// Mitsubishi GX Works2 project: BookEX6_39 Special Function   PLC: Q13UDV

// global labels: Global
VAR_GLOBAL
  bVar0 AT M5000 : BOOL;
  abArray0 AT M5010 : ARRAY [0..49] OF BOOL;
  sStr0 AT D5000 : STRING[199];
  sStr1 AT D5100 : STRING[199];
  sStr2 AT D5200 : STRING[199];
  sStr3 AT D5300 : STRING[199];
  sStr4 AT D5400 : STRING[199];
  sStr5 AT D5500 : STRING[199];
  sStr6 AT D5600 : STRING[199];
  sStr7 AT D5700 : STRING[199];
  sStr8 AT D5800 : STRING[199];
  sStr9 AT D5900 : STRING[199];
  iVar0 AT D4500 : INT;
  iVar1 AT D4501 : INT;
  iVar2 AT D4502 : INT;
  iVar3 AT D4503 : INT;
  iVar4 AT D4504 : INT;
  iVar5 AT D4505 : INT;
  iVar6 AT D4506 : INT;
  iVar7 AT D4507 : INT;
  iVar8 AT D4508 : INT;
  iVar9 AT D4509 : INT;
  dVar0 AT D4510 : DINT;
  dVar1 AT D4512 : DINT;
  dVar2 AT D4514 : DINT;
  dVar3 AT D4516 : DINT;
  dVar4 AT D4518 : DINT;
  dVar5 AT D4520 : DINT;
  dVar6 AT D4522 : DINT;
  dVar7 AT D4524 : DINT;
  dVar8 AT D4526 : DINT;
  dVar9 AT D4528 : DINT;
  wVar0 AT D4530 : WORD;
  wVar1 AT D4531 : WORD;
  wVar2 AT D4532 : WORD;
  wVar3 AT D4533 : WORD;
  wVar4 AT D4534 : WORD;
  wVar5 AT D4535 : WORD;
  wVar6 AT D4536 : WORD;
  wVar7 AT D4537 : WORD;
  wVar8 AT D4538 : WORD;
  wVar9 AT D4539 : WORD;
  dwVar0 AT D4540 : DWORD;
  dwVar1 AT D4542 : DWORD;
  dwVar2 AT D4544 : DWORD;
  dwVar3 AT D4546 : DWORD;
  dwVar4 AT D4548 : DWORD;
  dwVar5 AT D4550 : DWORD;
  dwVar6 AT D4552 : DWORD;
  dwVar7 AT D4554 : DWORD;
  dwVar8 AT D4556 : DWORD;
  dwVar9 AT D4558 : DWORD;
  fsVar0 AT D4560 : REAL;
  fsVar1 AT D4562 : REAL;
  fsVar2 AT D4564 : REAL;
  fsVar3 AT D4566 : REAL;
  fsVar4 AT D4568 : REAL;
  fsVar5 AT D4570 : REAL;
  fsVar6 AT D4572 : REAL;
  fsVar7 AT D4574 : REAL;
  fsVar8 AT D4576 : REAL;
  fsVar9 AT D4578 : REAL;
  fdVar0 AT D4580 : LREAL;
  tTime0 AT D4620 : TIME;
  tTime1 AT D4622 : TIME;
  tTime2 AT D4624 : TIME;
  tTime3 AT D4626 : TIME;
  tTime4 AT D4628 : TIME;
  tTime5 AT D4630 : TIME;
  tTime6 AT D4632 : TIME;
  tTime7 AT D4634 : TIME;
  tTime8 AT D4636 : TIME;
  tTime9 AT D4638 : TIME;
  tTime10 AT D4640 : TIME;
  bVar1 AT M5001 : BOOL;
  bVar2 AT M5002 : BOOL;
  bVar3 AT M5003 : BOOL;
  bVar4 AT M5004 : BOOL;
  bVar5 AT M5005 : BOOL;
  bVar6 AT M5006 : BOOL;
  bVar7 AT M5007 : BOOL;
  bVar8 AT M5008 : BOOL;
  bVar9 AT M5009 : BOOL;
  abArray1 AT M5060 : ARRAY [0..49] OF BOOL;
  abArray2 AT M5110 : ARRAY [0..49] OF BOOL;
  abArray3 AT M5160 : ARRAY [0..49] OF BOOL;
  abArray4 AT M5210 : ARRAY [0..49] OF BOOL;
  abArray5 AT M5260 : ARRAY [0..49] OF BOOL;
  abArray6 AT M5310 : ARRAY [0..49] OF BOOL;
  abArray7 AT M5360 : ARRAY [0..49] OF BOOL;
  abArray8 AT M5410 : ARRAY [0..49] OF BOOL;
  abArray9 AT M5460 : ARRAY [0..49] OF BOOL;
  fdVar1 AT D4584 : LREAL;
  fdVar2 AT D4588 : LREAL;
  fdVar3 AT D4592 : LREAL;
  fdVar4 AT D4596 : LREAL;
  fdVar5 AT D4600 : LREAL;
  fdVar6 AT D4604 : LREAL;
  fdVar7 AT D4608 : LREAL;
  fdVar8 AT D4612 : LREAL;
  fdVar9 AT D4616 : LREAL;
  afsPen0 AT D2000 : ARRAY [0..499] OF REAL;
  afsPen1 AT D3000 : ARRAY [0..499] OF REAL;
  adwD10 AT D10 : ARRAY [0..9] OF DWORD;
  awD10 AT D10 : ARRAY [0..19] OF WORD;
  aiD10 AT D10 : ARRAY [0..19] OF INT;
  abM10 AT M10 : ARRAY [0..19] OF BOOL;
END_VAR
// user libraries (not included): HMI

FUNCTION DEG2RAD
VAR_INPUT
  fs_Deg : REAL;
END_VAR
VAR
  fsTemp : REAL;
  fs2Phi : REAL;
  dFloor : DINT;
END_VAR
VAR CONSTANT
  Phi : REAL := 3.141592653;
END_VAR
;
fsTemp := 0.0174532925199433 * fs_Deg;
fs2Phi := Phi * 2.0;
dFloor := REAL_TO_DINT(fsTemp / fs2Phi );
Deg2Rad := fsTemp;
END_FUNCTION

FUNCTION_BLOCK GenLotto
VAR_OUTPUT
  i_Lotto1 : INT;
  i_Lotto2 : INT;
  i_Lotto3 : INT;
  i_Lotto4 : INT;
  i_Lotto5 : INT;
  i_Lotto6 : INT;
END_VAR
VAR
  fbGenRandom : GenRandom;
  ix : INT;
  iy : INT;
  aiNo : ARRAY [0..5] OF INT;
  aiSNo : ARRAY [0..1] OF INT;
  idx : INT;
  bSRes : BOOL;
  aiSNo1 : ARRAY [0..1] OF INT;
  dNo : DINT;
  iz : INT;
END_VAR
;
FOR ix := 0 TO 5 DO 
	aiNo[ix] := 0;
END_FOR;
idx := 0;

REPEAT
	fbGenRandom(EN := TRUE, d_Low := 1, d_High := 45);
	dNo := fbGenRandom.d_Out;
	iy := DINT_TO_INT(dNo);
	SER(TRUE, iy, aiNo[0], 6, aiSNo);
	IF aiSNo[1] = 0 THEN
		aiNo[idx] := iy;
		idx := idx + 1;
	END_IF;
	UNTIL idx > 5
END_REPEAT;	
(* Sort *)
FOR ix := 0 TO 4 DO 
	FOR iy := 0 TO 4 DO 
		IF aiNo[iy] > aiNo[iy+1] THEN
			iz := aiNo[iy];
			aiNo[iy] := aiNo[iy+1];
			aiNo[iy+1] := iz;
		END_IF;
	END_FOR;
END_FOR;

i_Lotto1 := aiNo[0];
i_Lotto2 := aiNo[1];
i_Lotto3 := aiNo[2];
i_Lotto4 := aiNo[3];
i_Lotto5 := aiNo[4];
i_Lotto6 := aiNo[5];
END_FUNCTION_BLOCK

FUNCTION_BLOCK GenRandom
VAR_INPUT
  d_Low : DINT;
  d_High : DINT;
END_VAR
VAR
  dwTemp1 : DWORD;
END_VAR
VAR_OUTPUT
  d_Out : DINT;
END_VAR
VAR
  dLast : DINT;
  iTime : ARRAY [0..7] OF INT;
  dwTemp2 : DWORD;
  dwTemp3 : DWORD;
END_VAR
;
S_DATERD(TRUE, iTime);
dwTemp1 := DINT_TO_DWORD(INT_TO_DINT(iTime[5]) * 10000 + INT_TO_DINT(iTime[6]) * 1000 + INT_TO_DINT(iTime[7]));
dwTemp2 := SHL(dwTemp1, 15) XOR dwTemp1;
dwTemp2 := SHL(dwTemp2, 13) XOR dwTemp2;
dwTemp2 := SHR(dwTemp2, 17) XOR dwTemp2;
dLast := DWORD_TO_DINT(SHL(dwTemp2, 5) XOR dwTemp2);
d_Out := ABS(dLast MOD (d_High - d_Low + 1)) + d_Low;
END_FUNCTION_BLOCK

FUNCTION_BLOCK GenWave
VAR_INPUT
  t_Period : TIME;
  dDelay : DINT;  (* % *)
  fs_Amp : REAL;
  fs_Offset : REAL;
END_VAR
VAR_OUTPUT
  b_Q : BOOL;
  i_OutV : INT;
END_VAR
VAR
  fsTemp : REAL;
  fsTemp1 : REAL;
  tLast : TIME;
  tPast : TIME;
  tCurr : TIME;
  tMulTime : TIME;
  tShift : TIME;
  dSftTime : DINT;
  bInit : BOOL;
  qTemp : BOOL;
END_VAR
VAR CONSTANT
  PI2 : REAL := 6.283185;
END_VAR
VAR
  fbTON : TON;
END_VAR
VAR_INPUT
  i_Type : INT;
END_VAR
VAR
  dMulTime : DINT;
  dHalfPeriod : DINT;
END_VAR
;
fbTON(IN := NOT qTemp, PT := T#30m, Q:= qTemp, ET := tPast);
tCurr := tPast - tLast;

IF NOT bInit THEN
	bInit := TRUE;
	tLast := tCurr;
	tCurr := T#0s;
END_IF;

IF tCurr >= t_Period THEN
	tLast := tLast + t_Period;
	tCurr := tCurr - t_Period;
END_IF;

CASE i_Type OF 
	0 : (* SIN *)
		IF t_Period > T#0s THEN
			dSftTime := TIME_TO_DINT(t_Period) * dDelay / 100;
			tShift := DINT_TO_TIME(dSftTime);
			tMulTime := tCurr - tShift;
			fsTemp1 := PI2 * DINT_TO_REAL(TIME_TO_DINT(tMulTime)) / DINT_TO_REAL(TIME_TO_DINT(t_Period));
			SIN(TRUE, fsTemp1, fsTemp);
		ELSE
			fsTemp := 0.0;
		END_IF;
	1 : (* SQUARE *)
		IF t_Period > T#0s THEN
			dMulTime := TIME_TO_DINT(tCurr);
			dHalfPeriod := TIME_TO_DINT(t_Period) / 2;
			IF dMulTime < dHalfPeriod THEN
				fsTemp := 1.0;
			ELSE
				fsTemp := -1.0;
			END_IF;
		ELSE
			fsTemp := 0.0;
		END_IF; 
	2 : (* SAW *)
		IF t_Period > T#0s THEN
			fsTemp := DINT_TO_REAL(TIME_TO_DINT(tCurr) * 2) / DINT_TO_REAL(TIME_TO_DINT(t_Period)) - 1.0;
		ELSE
			fsTemp := 0.0;
		END_IF;
END_CASE;
i_OutV := REAL_TO_INT(fs_Amp * fsTemp * 0.5  + fs_Offset);
b_Q := i_OutV < 0;
END_FUNCTION_BLOCK

FUNCTION RAD2DEG
VAR_INPUT
  fs_Rad : REAL;
END_VAR
VAR
  fsTemp : REAL;
  fs2Phi : REAL;
  dFloor : DINT;
END_VAR
VAR CONSTANT
  Phi : REAL := 3.141592653;
END_VAR
;
fsTemp := 57.29577951308232 * fs_Rad;
dFloor := REAL_TO_DINT(fsTemp / 360.0);
Rad2Deg := fsTemp;
END_FUNCTION

PROGRAM ExASIN
VAR
  awBCD1 : ARRAY [0..2] OF WORD;
  Mov4WORD_1 : Mov4WORD;
  Mov4WORD_2 : Mov4WORD;
  Mov4WORD_3 : Mov4WORD;
  awBCD2 : ARRAY [0..2] OF WORD;
  awBCD3 : ARRAY [0..2] OF WORD;
  Mov4WORD_4 : Mov4WORD;
  awBCD4 : ARRAY [0..2] OF WORD;
  awBCD5 : ARRAY [0..2] OF WORD;
END_VAR
(* structured ladder/FBD written out as ST: instructions are called as NAME(EN, inputs, outputs); _pN, _eN, _tN stand for wires *)
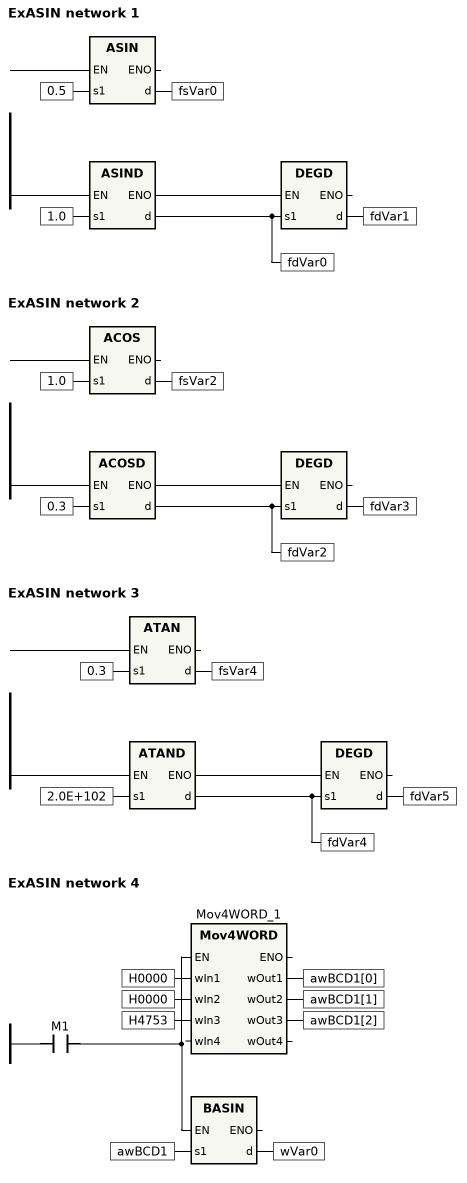
(* network 1 *)
ASIN(TRUE, 0.5, fsVar0);
_e1 := ASIND(TRUE, 1.0, fdVar0);
DEGD(_e1, fdVar0, fdVar1);
(* network 2 *)
ACOS(TRUE, 1.0, fsVar2);
_e1 := ACOSD(TRUE, 0.3, fdVar2);
DEGD(_e1, fdVar2, fdVar3);
(* network 3 *)
ATAN(TRUE, 0.3, fsVar4);
_e1 := ATAND(TRUE, 2.0E+102, fdVar4);
DEGD(_e1, fdVar4, fdVar5);
(* network 4 *)
Mov4WORD_1(EN := M1, wIn1 := H0000, wIn2 := H0000, wIn3 := H4753, wOut1 => awBCD1[0], wOut2 => awBCD1[1], wOut3 => awBCD1[2]);
BASIN(M1, awBCD1, wVar0);
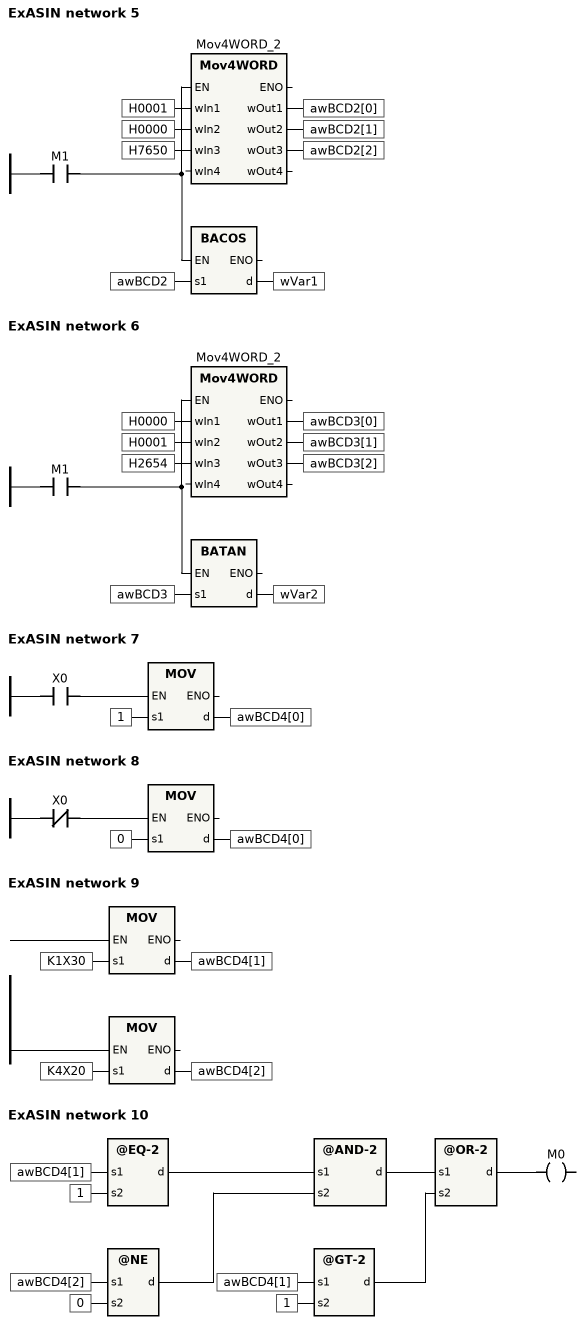
(* network 5 *)
Mov4WORD_2(EN := M1, wIn1 := H0001, wIn2 := H0000, wIn3 := H7650, wOut1 => awBCD2[0], wOut2 => awBCD2[1], wOut3 => awBCD2[2]);
BACOS(M1, awBCD2, wVar1);
(* network 6 *)
Mov4WORD_2(EN := M1, wIn1 := H0000, wIn2 := H0001, wIn3 := H2654, wOut1 => awBCD3[0], wOut2 => awBCD3[1], wOut3 => awBCD3[2]);
BATAN(M1, awBCD3, wVar2);
(* network 7 *)
MOV(X0, 1, awBCD4[0]);
(* network 8 *)
MOV(NOT X0, 0, awBCD4[0]);
(* network 9 *)
MOV(TRUE, K1X30, awBCD4[1]);
MOV(TRUE, K4X20, awBCD4[2]);
(* network 10 *)
M0 := @OR-2(@AND-2(@EQ-2(awBCD4[1], 1), @NE(awBCD4[2], 0)), @GT-2(awBCD4[1], 1));
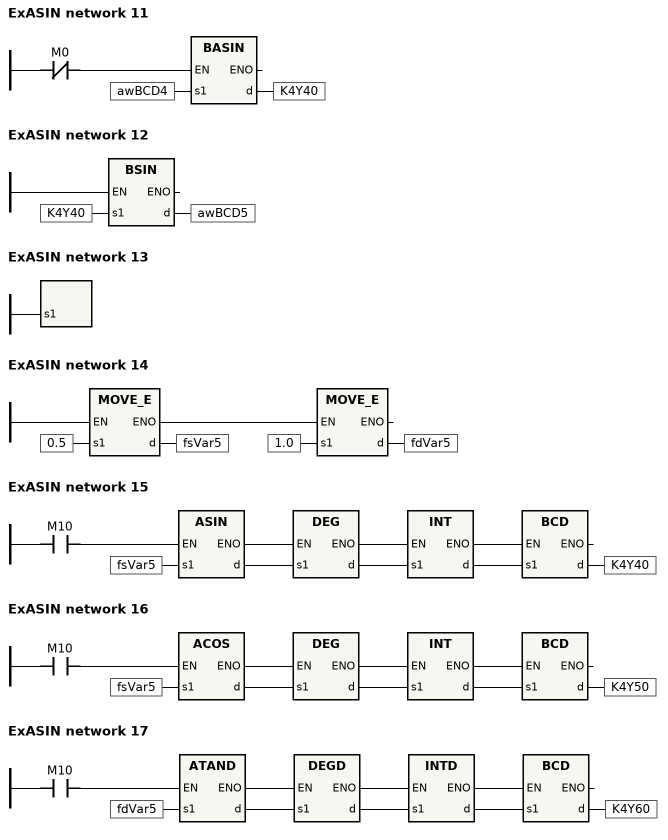
(* network 11 *)
BASIN(NOT M0, awBCD4, K4Y40);
(* network 12 *)
BSIN(TRUE, K4Y40, awBCD5);
(* network 13 *)
(* element kind 10  <- TRUE *)
(* network 14 *)
_e1 := MOVE_E(TRUE, 0.5, fsVar5);
MOVE_E(_e1, 1.0, fdVar5);
(* network 15 *)
_e2 := ASIN(M10, fsVar5, _t1);
_e4 := DEG(_e2, _t1, _t3);
_e6 := INT(_e4, _t3, _t5);
BCD(_e6, _t5, K4Y40);
(* network 16 *)
_e2 := ACOS(M10, fsVar5, _t1);
_e4 := DEG(_e2, _t1, _t3);
_e6 := INT(_e4, _t3, _t5);
BCD(_e6, _t5, K4Y50);
(* network 17 *)
_e2 := ATAND(M10, fdVar5, _t1);
_e4 := DEGD(_e2, _t1, _t3);
_e6 := INTD(_e4, _t3, _t5);
BCD(_e6, _t5, K4Y60);
END_PROGRAM

PROGRAM ExDEG_RAD
VAR
  fsLVar0 : REAL;
  fsLVar1 : REAL;
  fsLVar2 : REAL;
  fsLVar3 : REAL;
  fsLVar4 : REAL;
  fsLVar5 : REAL;
  fsLVar6 : REAL;
  fsLVar7 : REAL;
  fsLVar8 : REAL;
  fsLVar9 : REAL;
END_VAR
(* structured ladder/FBD written out as ST: instructions are called as NAME(EN, inputs, outputs); _pN, _eN, _tN stand for wires *)
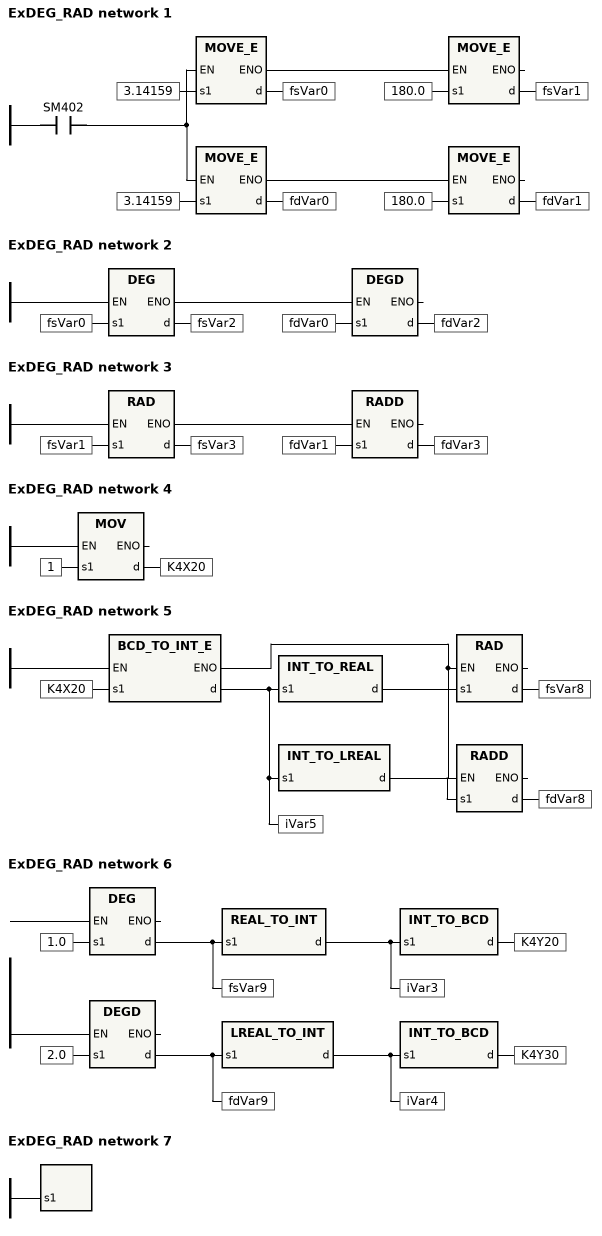
(* network 1 *)
_e1 := MOVE_E(SM402, 3.14159, fsVar0);
MOVE_E(_e1, 180.0, fsVar1);
_e2 := MOVE_E(SM402, 3.14159, fdVar0);
MOVE_E(_e2, 180.0, fdVar1);
(* network 2 *)
_e1 := DEG(TRUE, fsVar0, fsVar2);
DEGD(_e1, fdVar0, fdVar2);
(* network 3 *)
_e1 := RAD(TRUE, fsVar1, fsVar3);
RADD(_e1, fdVar1, fdVar3);
(* network 4 *)
MOV(TRUE, 1, K4X20);
(* network 5 *)
_e1 := BCD_TO_INT_E(TRUE, K4X20, iVar5);
RAD(_e1, INT_TO_REAL(iVar5), fsVar8);
RADD(_e1, INT_TO_LREAL(iVar5), fdVar8);
(* network 6 *)
DEG(TRUE, 1.0, fsVar9);
_p1 := REAL_TO_INT(fsVar9);
iVar3 := _p1;
K4Y20 := INT_TO_BCD(_p1);
DEGD(TRUE, 2.0, fdVar9);
_p2 := LREAL_TO_INT(fdVar9);
iVar4 := _p2;
K4Y30 := INT_TO_BCD(_p2);
(* network 7 *)
(* element kind 10  <- TRUE *)
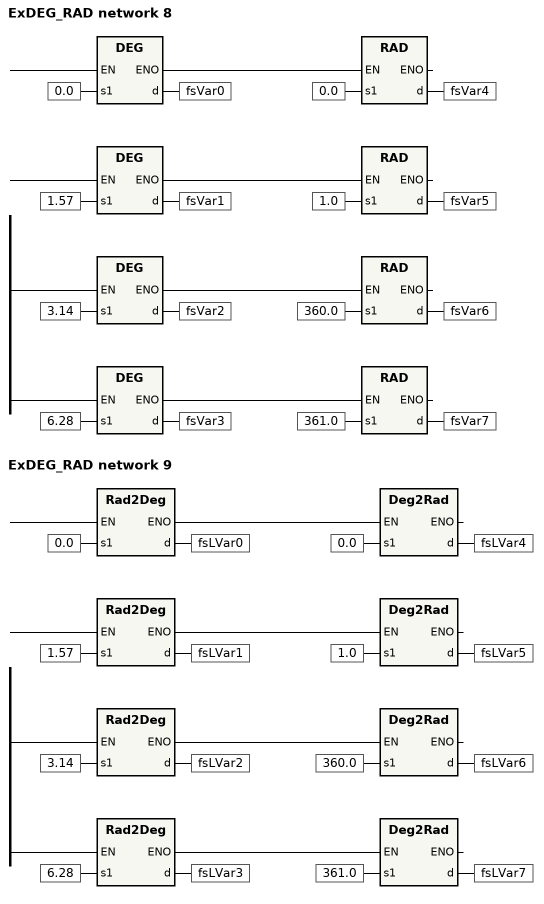
(* network 8 *)
_e1 := DEG(TRUE, 0.0, fsVar0);
RAD(_e1, 0.0, fsVar4);
_e2 := DEG(TRUE, 1.57, fsVar1);
RAD(_e2, 1.0, fsVar5);
_e3 := DEG(TRUE, 3.14, fsVar2);
RAD(_e3, 360.0, fsVar6);
_e4 := DEG(TRUE, 6.28, fsVar3);
RAD(_e4, 361.0, fsVar7);
(* network 9 *)
_e1 := Rad2Deg(TRUE, 0.0, fsLVar0);
Deg2Rad(_e1, 0.0, fsLVar4);
_e2 := Rad2Deg(TRUE, 1.57, fsLVar1);
Deg2Rad(_e2, 1.0, fsLVar5);
_e3 := Rad2Deg(TRUE, 3.14, fsLVar2);
Deg2Rad(_e3, 360.0, fsLVar6);
_e4 := Rad2Deg(TRUE, 6.28, fsLVar3);
Deg2Rad(_e4, 361.0, fsLVar7);
END_PROGRAM

PROGRAM ExEXP
(* structured ladder/FBD written out as ST: instructions are called as NAME(EN, inputs, outputs); _pN, _eN, _tN stand for wires *)
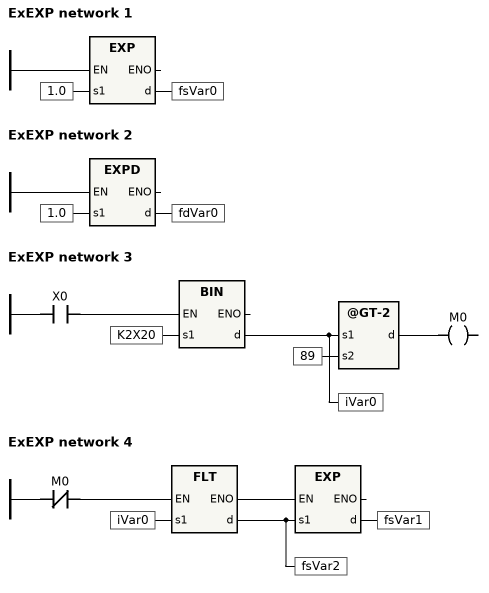
(* network 1 *)
EXP(TRUE, 1.0, fsVar0);
(* network 2 *)
EXPD(TRUE, 1.0, fdVar0);
(* network 3 *)
BIN(X0, K2X20, iVar0);
M0 := @GT-2(iVar0, 89);
(* network 4 *)
_e1 := FLT(NOT M0, iVar0, fsVar2);
EXP(_e1, fsVar2, fsVar1);
END_PROGRAM

PROGRAM ExGetWave
VAR
  GenWave_1 : GenWave;
  GenWave_2 : GenWave;
  GenWave_3 : GenWave;
  GenWave_4 : GenWave;
END_VAR
(* structured ladder/FBD written out as ST: instructions are called as NAME(EN, inputs, outputs); _pN, _eN, _tN stand for wires *)
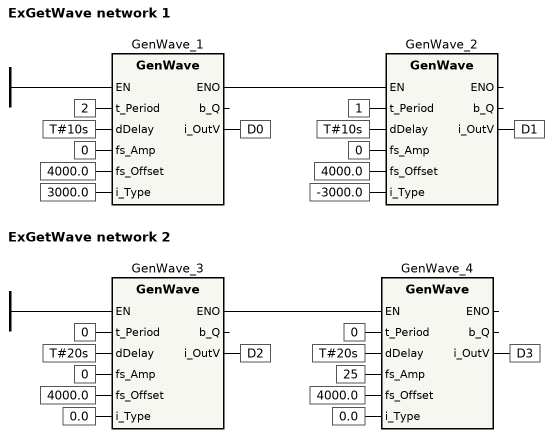
(* network 1 *)
GenWave_1(EN := TRUE, t_Period := 2, dDelay := T#10s, fs_Amp := 0, fs_Offset := 4000.0, i_Type := 3000.0, i_OutV => D0);
GenWave_2(EN := GenWave_1.ENO, t_Period := 1, dDelay := T#10s, fs_Amp := 0, fs_Offset := 4000.0, i_Type := -3000.0, i_OutV => D1);
(* network 2 *)
GenWave_3(EN := TRUE, t_Period := 0, dDelay := T#20s, fs_Amp := 0, fs_Offset := 4000.0, i_Type := 0.0, i_OutV => D2);
GenWave_4(EN := GenWave_3.ENO, t_Period := 0, dDelay := T#20s, fs_Amp := 25, fs_Offset := 4000.0, i_Type := 0.0, i_OutV => D3);
END_PROGRAM

PROGRAM ExLOG
(* structured ladder/FBD written out as ST: instructions are called as NAME(EN, inputs, outputs); _pN, _eN, _tN stand for wires *)
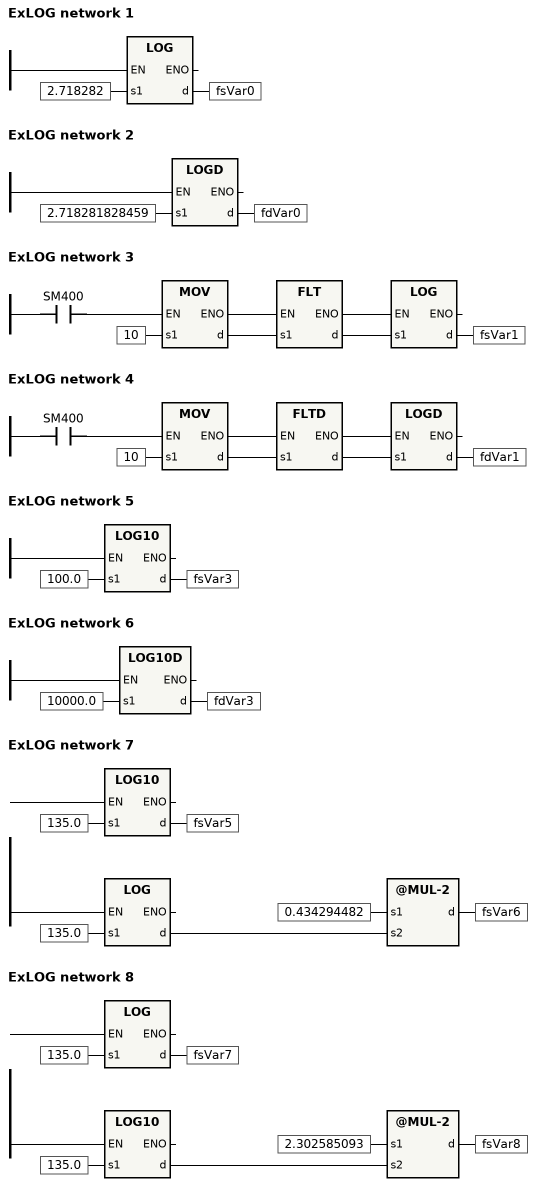
(* network 1 *)
LOG(TRUE, 2.718282, fsVar0);
(* network 2 *)
LOGD(TRUE, 2.718281828459, fdVar0);
(* network 3 *)
_e2 := MOV(SM400, 10, _t1);
_e4 := FLT(_e2, _t1, _t3);
LOG(_e4, _t3, fsVar1);
(* network 4 *)
_e2 := MOV(SM400, 10, _t1);
_e4 := FLTD(_e2, _t1, _t3);
LOGD(_e4, _t3, fdVar1);
(* network 5 *)
LOG10(TRUE, 100.0, fsVar3);
(* network 6 *)
LOG10D(TRUE, 10000.0, fdVar3);
(* network 7 *)
LOG10(TRUE, 135.0, fsVar5);
LOG(TRUE, 135.0, _t1);
fsVar6 := @MUL-2(0.434294482, _t1);
(* network 8 *)
LOG(TRUE, 135.0, fsVar7);
LOG10(TRUE, 135.0, _t1);
fsVar8 := @MUL-2(2.302585093, _t1);
END_PROGRAM

PROGRAM ExPOW
(* structured ladder/FBD written out as ST: instructions are called as NAME(EN, inputs, outputs); _pN, _eN, _tN stand for wires *)
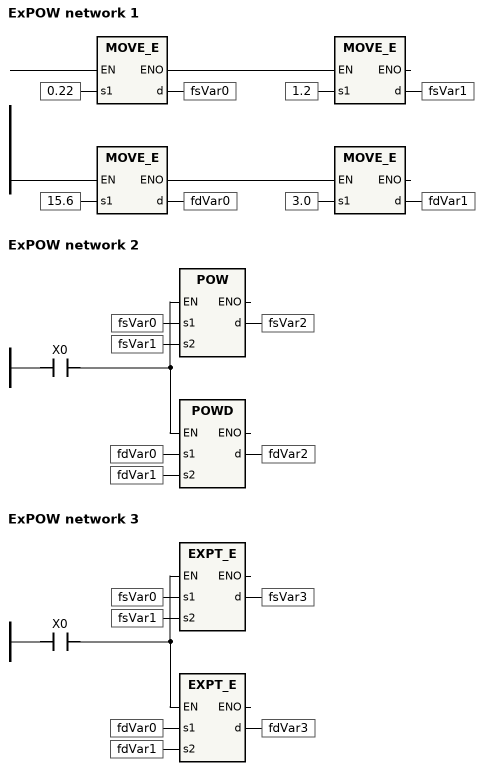
(* network 1 *)
_e1 := MOVE_E(TRUE, 0.22, fsVar0);
MOVE_E(_e1, 1.2, fsVar1);
_e2 := MOVE_E(TRUE, 15.6, fdVar0);
MOVE_E(_e2, 3.0, fdVar1);
(* network 2 *)
POW(X0, fsVar0, fsVar1, fsVar2);
POWD(X0, fdVar0, fdVar1, fdVar2);
(* network 3 *)
EXPT_E(X0, fsVar0, fsVar1, fsVar3);
EXPT_E(X0, fdVar0, fdVar1, fdVar3);
END_PROGRAM

PROGRAM ExRAD
(* structured ladder/FBD written out as ST: instructions are called as NAME(EN, inputs, outputs); _pN, _eN, _tN stand for wires *)
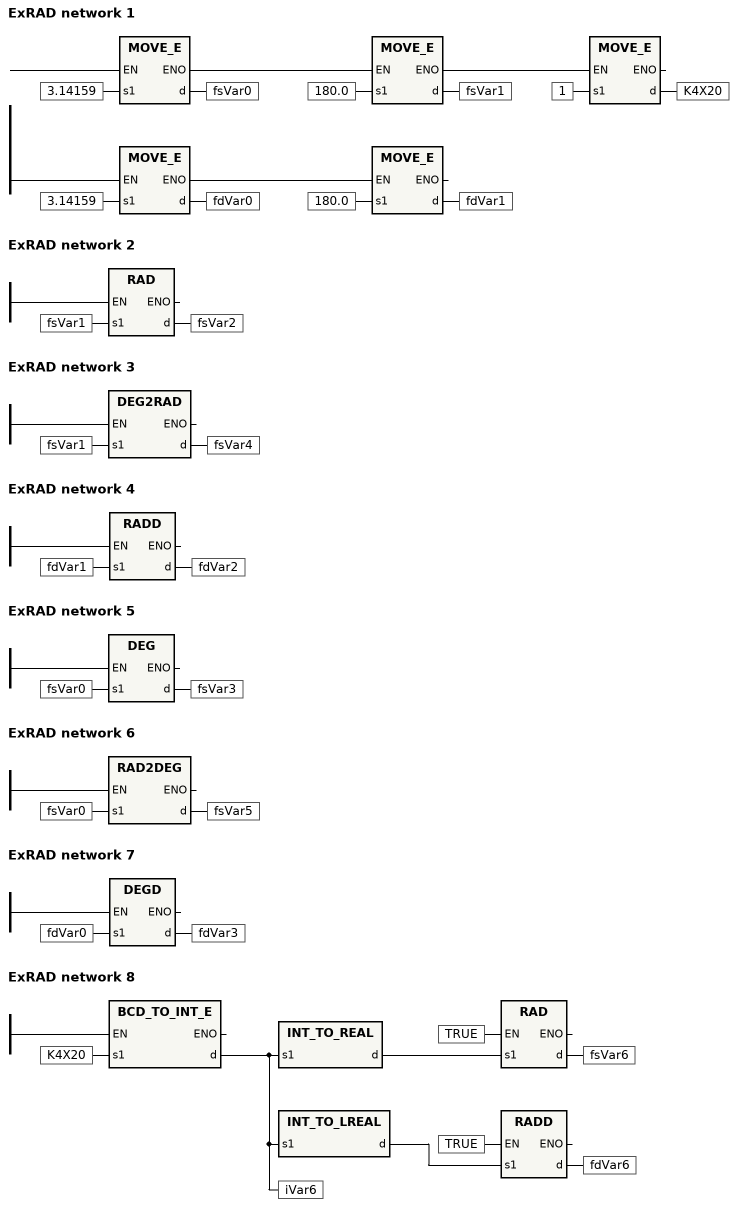
(* network 1 *)
_e1 := MOVE_E(TRUE, 3.14159, fsVar0);
_e2 := MOVE_E(_e1, 180.0, fsVar1);
MOVE_E(_e2, 1, K4X20);
_e3 := MOVE_E(TRUE, 3.14159, fdVar0);
MOVE_E(_e3, 180.0, fdVar1);
(* network 2 *)
RAD(TRUE, fsVar1, fsVar2);
(* network 3 *)
DEG2RAD(TRUE, fsVar1, fsVar4);
(* network 4 *)
RADD(TRUE, fdVar1, fdVar2);
(* network 5 *)
DEG(TRUE, fsVar0, fsVar3);
(* network 6 *)
RAD2DEG(TRUE, fsVar0, fsVar5);
(* network 7 *)
DEGD(TRUE, fdVar0, fdVar3);
(* network 8 *)
BCD_TO_INT_E(TRUE, K4X20, iVar6);
RAD(TRUE, INT_TO_REAL(iVar6), fsVar6);
RADD(TRUE, INT_TO_LREAL(iVar6), fdVar6);
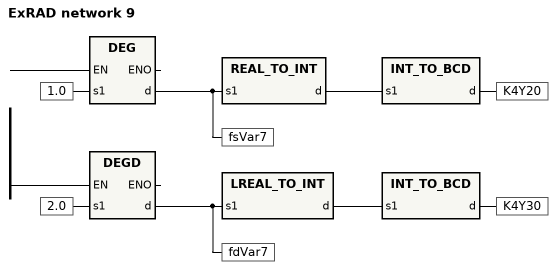
(* network 9 *)
DEG(TRUE, 1.0, fsVar7);
K4Y20 := INT_TO_BCD(REAL_TO_INT(fsVar7));
DEGD(TRUE, 2.0, fdVar7);
K4Y30 := INT_TO_BCD(LREAL_TO_INT(fdVar7));
END_PROGRAM

PROGRAM ExRND
VAR
  CurrTime : ARRAY [0..7] OF INT;
  GenRandom_1 : GenRandom;
  GenRandom_2 : GenRandom;
  GenRandom_3 : GenRandom;
  GenRandom_4 : GenRandom;
  GenRandom_5 : GenRandom;
  GenRandom_6 : GenRandom;
  GenLotto_1 : GenLotto;
END_VAR
(* structured ladder/FBD written out as ST: instructions are called as NAME(EN, inputs, outputs); _pN, _eN, _tN stand for wires *)
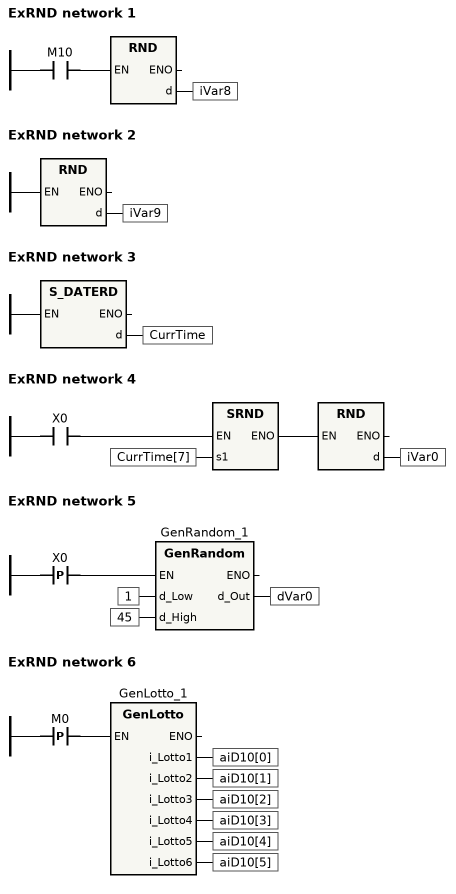
(* network 1 *)
RND(M10, iVar8);
(* network 2 *)
RND(TRUE, iVar9);
(* network 3 *)
S_DATERD(TRUE, CurrTime);
(* network 4 *)
_e1 := SRND(X0, CurrTime[7]);
RND(_e1, iVar0);
(* network 5 *)
GenRandom_1(EN := LDP(TRUE, X0), d_Low := 1, d_High := 45, d_Out => dVar0);
(* network 6 *)
GenLotto_1(EN := LDP(TRUE, M0), i_Lotto1 => aiD10[0], i_Lotto2 => aiD10[1], i_Lotto3 => aiD10[2], i_Lotto4 => aiD10[3], i_Lotto5 => aiD10[4], i_Lotto6 => aiD10[5]);
END_PROGRAM

PROGRAM ExSIN
VAR
  awBCD1 : ARRAY [0..2] OF WORD;
  Mov4WORD_1 : Mov4WORD;
  Mov4WORD_2 : Mov4WORD;
  Mov4WORD_3 : Mov4WORD;
  awBCD2 : ARRAY [0..2] OF WORD;
  awBCD3 : ARRAY [0..2] OF WORD;
  Mov4WORD_4 : Mov4WORD;
  awBCD4 : ARRAY [0..2] OF WORD;
  aw2BCD : ARRAY [0..1] OF WORD;
END_VAR
(* structured ladder/FBD written out as ST: instructions are called as NAME(EN, inputs, outputs); _pN, _eN, _tN stand for wires *)
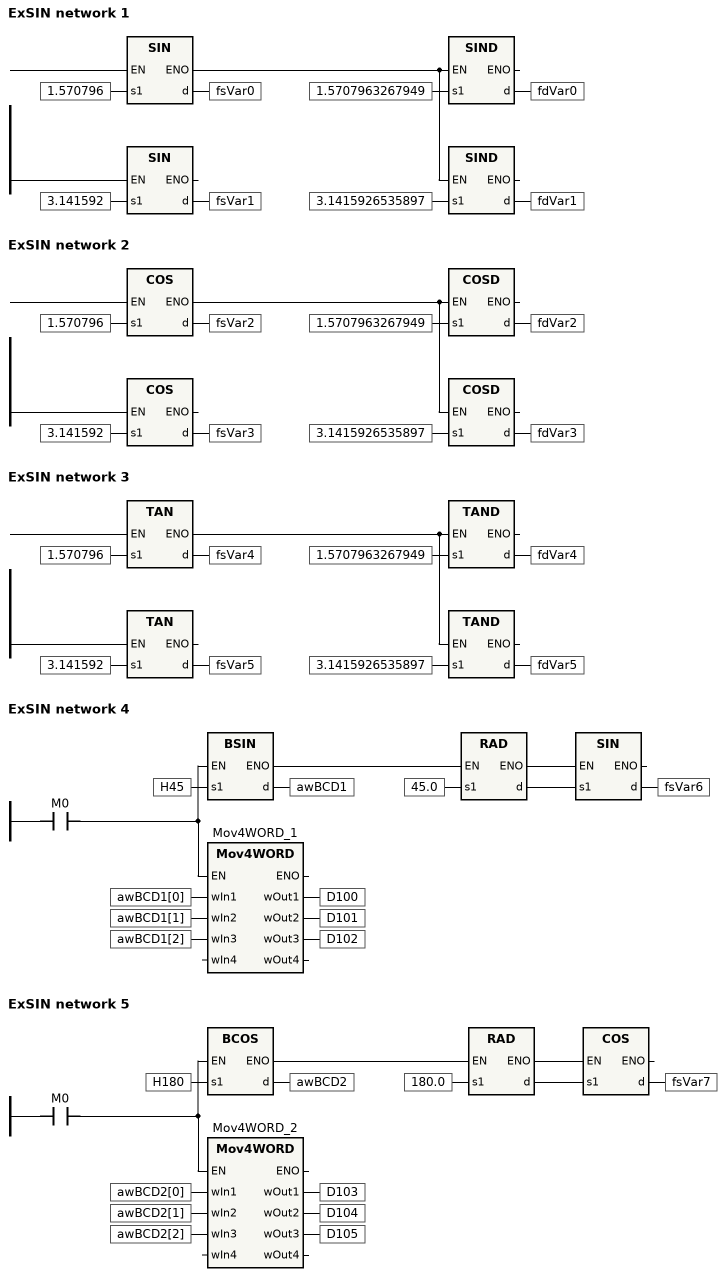
(* network 1 *)
_e1 := SIN(TRUE, 1.570796, fsVar0);
SIND(_e1, 1.5707963267949, fdVar0);
SIN(TRUE, 3.141592, fsVar1);
SIND(_e1, 3.1415926535897, fdVar1);
(* network 2 *)
_e1 := COS(TRUE, 1.570796, fsVar2);
COSD(_e1, 1.5707963267949, fdVar2);
COS(TRUE, 3.141592, fsVar3);
COSD(_e1, 3.1415926535897, fdVar3);
(* network 3 *)
_e1 := TAN(TRUE, 1.570796, fsVar4);
TAND(_e1, 1.5707963267949, fdVar4);
TAN(TRUE, 3.141592, fsVar5);
TAND(_e1, 3.1415926535897, fdVar5);
(* network 4 *)
_e1 := BSIN(M0, H45, awBCD1);
_e3 := RAD(_e1, 45.0, _t2);
SIN(_e3, _t2, fsVar6);
Mov4WORD_1(EN := M0, wIn1 := awBCD1[0], wIn2 := awBCD1[1], wIn3 := awBCD1[2], wOut1 => D100, wOut2 => D101, wOut3 => D102);
(* network 5 *)
_e1 := BCOS(M0, H180, awBCD2);
_e3 := RAD(_e1, 180.0, _t2);
COS(_e3, _t2, fsVar7);
Mov4WORD_2(EN := M0, wIn1 := awBCD2[0], wIn2 := awBCD2[1], wIn3 := awBCD2[2], wOut1 => D103, wOut2 => D104, wOut3 => D105);
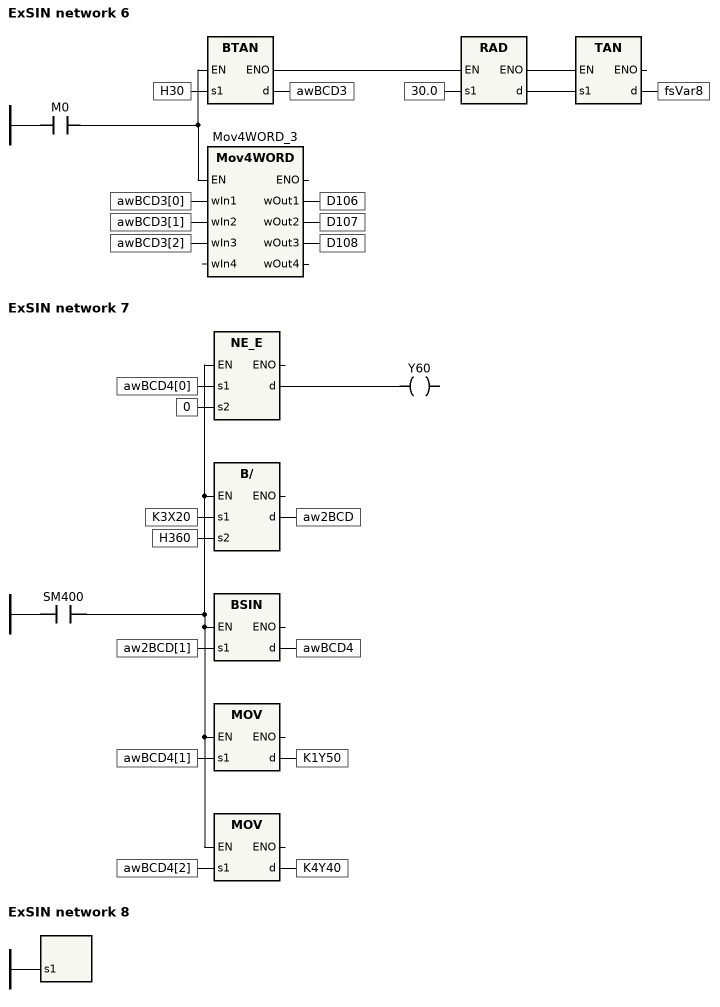
(* network 6 *)
_e1 := BTAN(M0, H30, awBCD3);
_e3 := RAD(_e1, 30.0, _t2);
TAN(_e3, _t2, fsVar8);
Mov4WORD_3(EN := M0, wIn1 := awBCD3[0], wIn2 := awBCD3[1], wIn3 := awBCD3[2], wOut1 => D106, wOut2 => D107, wOut3 => D108);
(* network 7 *)
B/(SM400, K3X20, H360, aw2BCD);
BSIN(SM400, aw2BCD[1], awBCD4);
MOV(SM400, awBCD4[1], K1Y50);
MOV(SM400, awBCD4[2], K4Y40);
NE_E(SM400, awBCD4[0], 0, _t1);
Y60 := _t1;
(* network 8 *)
(* element kind 10  <- TRUE *)
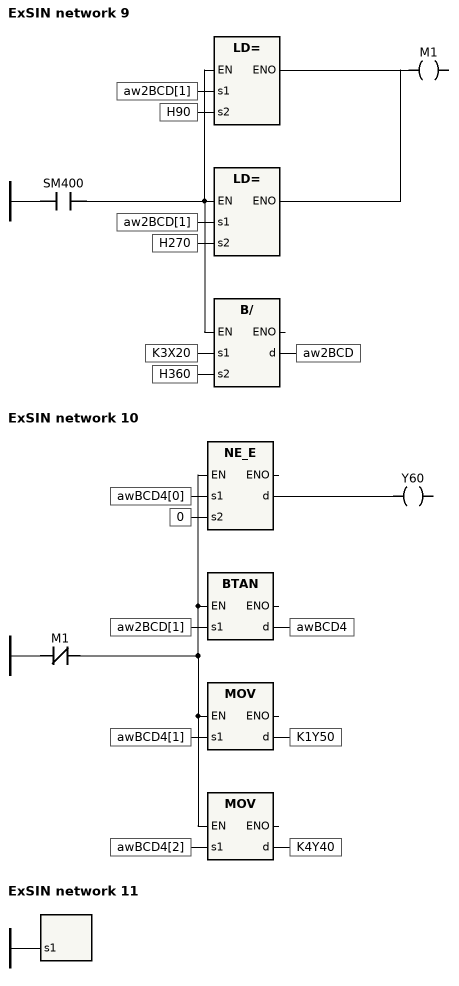
(* network 9 *)
B/(SM400, K3X20, H360, aw2BCD);
_e1 := LD=(SM400, aw2BCD[1], H90);
_e2 := LD=(SM400, aw2BCD[1], H270);
M1 := _e1 OR _e2;
(* network 10 *)
_p1 := NOT M1;
BTAN(_p1, aw2BCD[1], awBCD4);
MOV(_p1, awBCD4[1], K1Y50);
MOV(_p1, awBCD4[2], K4Y40);
NE_E(_p1, awBCD4[0], 0, _t2);
Y60 := _t2;
(* network 11 *)
(* element kind 10  <- TRUE *)
END_PROGRAM

PROGRAM ExSinGraph
VAR
  ix : INT;
  radx : REAL;
  fsx1 : REAL;
  fsx2 : REAL;
END_VAR
 
CASE iVar0 OF 
	0 : (* SIN *)
		fsVar8 := -1.0;		 (* MIN *)
		fsVar9 := 1.0;		 (* MAX *)	
		FOR ix := 0 TO 359 DO
			afsPen0[ix] := INT_TO_REAL(ix);
			RAD(TRUE,INT_TO_REAL(ix),radx);
			SIN(TRUE, radx, fsx2);
			afsPen1[ix] := fsx2;
		END_FOR;
 	1 : (* COS *)
		fsVar8 := -1.0;		 (* MIN *)
		fsVar9 := 1.0;		 (* MAX *)	
		FOR ix := 0 TO 359 DO
			afsPen0[ix] := INT_TO_REAL(ix);
			RAD(TRUE,INT_TO_REAL(ix),radx);
			COS(TRUE, radx, fsx2);
			afsPen1[ix] := fsx2;
		END_FOR;
 	2 : (* TAN *)
		fsVar8 := -10.0;		 (* MIN *)
		fsVar9 := 10.0;		 (* MAX *)	
		FOR ix := 0 TO 359 DO
			afsPen0[ix] := INT_TO_REAL(ix);
			RAD(TRUE,INT_TO_REAL(ix),radx);
			TAN(TRUE, radx, fsx2);
			afsPen1[ix] := fsx2;
		END_FOR;
END_CASE;
END_PROGRAM

PROGRAM ExSQR
VAR
  awRes : ARRAY [0..1] OF WORD;
  awRes2 : ARRAY [0..1] OF WORD;
END_VAR
(* structured ladder/FBD written out as ST: instructions are called as NAME(EN, inputs, outputs); _pN, _eN, _tN stand for wires *)
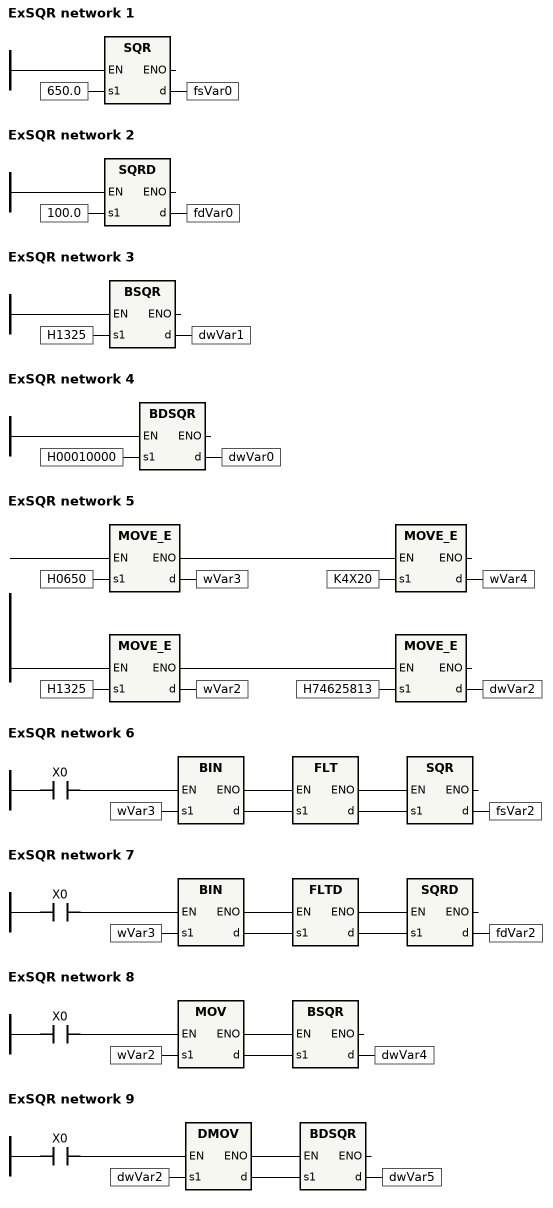
(* network 1 *)
SQR(TRUE, 650.0, fsVar0);
(* network 2 *)
SQRD(TRUE, 100.0, fdVar0);
(* network 3 *)
BSQR(TRUE, H1325, dwVar1);
(* network 4 *)
BDSQR(TRUE, H00010000, dwVar0);
(* network 5 *)
_e1 := MOVE_E(TRUE, H0650, wVar3);
MOVE_E(_e1, K4X20, wVar4);
_e2 := MOVE_E(TRUE, H1325, wVar2);
MOVE_E(_e2, H74625813, dwVar2);
(* network 6 *)
_e2 := BIN(X0, wVar3, _t1);
_e4 := FLT(_e2, _t1, _t3);
SQR(_e4, _t3, fsVar2);
(* network 7 *)
_e2 := BIN(X0, wVar3, _t1);
_e4 := FLTD(_e2, _t1, _t3);
SQRD(_e4, _t3, fdVar2);
(* network 8 *)
_e2 := MOV(X0, wVar2, _t1);
BSQR(_e2, _t1, dwVar4);
(* network 9 *)
_e2 := DMOV(X0, dwVar2, _t1);
BDSQR(_e2, _t1, dwVar5);
END_PROGRAM
